TYPE ST_Fan_op :
STRUCT
	OnOff	 	AT%Q* : BOOL;
	Speed		AT%Q* : INT;
END_STRUCT
END_TYPE

(* stored: Version 1.1.0.1, ProductVersion 3.1.4024.12
   DUT ST_Fan_op: Id {ec675ce8-f31a-48bb-b668-11dc399b90ed} *)
